FUNCTION_BLOCK REAL_ARRAY (* Tamplate for a simple Basic Function Block Type *)
  (* Standard: 61499-2 *)
  (* Version 0.0, 2019-03-10, 4DIAC-IDE, 4DIAC-Consortium *)
  (* Version 1.0, 2016-05-26, AZ, fortiss GmbH *)
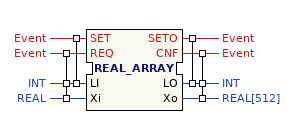
  EVENT_INPUT
    SET WITH LI; (* Trigger for Sending Array length *)
    REQ WITH LI, Xi; (* Normal Execution Request *)
  END_EVENT
  EVENT_OUTPUT
    SETO WITH LO; (* Sending event for Setting Array length *)
    CNF WITH LO, Xo; (* Confirmation of Execution *)
  END_EVENT
  VAR_INPUT
    LI : INT; (* Array length *)
    Xi : REAL; (* Input real component *)
  END_VAR
  VAR_OUTPUT
    LO : INT; (* Array length *)
    Xo : ARRAY [0..511] OF REAL; (* Output real array *)
  END_VAR
  VAR
    L : INT; (* Array length *)
    a : INT; (* Index of array *)
  END_VAR
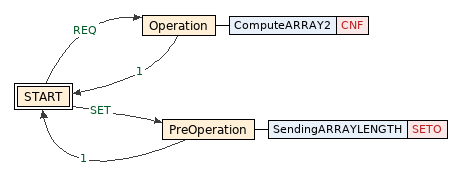
  EC_STATES
    START; (* Initial State *)
    Operation : ComputeARRAY2 -> CNF;
    PreOperation : SendingARRAYLENGTH -> SETO;
  END_STATES
  EC_TRANSITIONS
    START TO Operation := REQ;
    Operation TO START := 1;
    START TO PreOperation := SET;
    PreOperation TO START := 1;
  END_TRANSITIONS
  ALGORITHM ComputeARRAY2 IN ST: (* new algorithm *)
L := LI;
for a := 1 to L-1 do
	Xo[ a -1 ] := Xo[ a ]; //menggeser slot array
end_for;
Xo[ L - 1 ] := Xi; // memasukan nilai
LO := L; //cuma menunjukkan
  END_ALGORITHM
  ALGORITHM SendingARRAYLENGTH IN ST: (* new algorithm *)
LO := LI;
  END_ALGORITHM
END_FUNCTION_BLOCK
